% RSLogix 500 project Lab1 SLC500 3.RSS, saved by version 8.30.00.16 %
PROJECT "UNTITLED"    % processor: Bul.1763 MicroLogix 1100 Series B %

PROGRAM FILES
  LAD 2   3 rungs

DATA FILES
  O0 OUTPUT  4 elements
  I1 INPUT  6 elements
  S2 STATUS  66 elements
  B3 BINARY  1 elements
  T4 TIMER  1 elements
  C5 COUNTER  1 elements
  R6 CONTROL  1 elements
  N7 INTEGER  1 elements
  F8 FLOAT  1 elements

LADDER 2
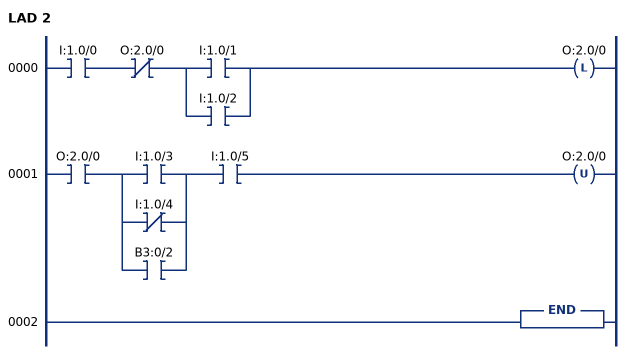
% Rung: 0 %  % edit flag set %
SOR XIC I:1.0/0 XIO O:2.0/0 BST XIC I:1.0/1 NXB XIC I:1.0/2 BND OTL O:2.0/0 EOR
% Rung: 1 %  % edit flag set %
SOR XIC O:2.0/0 BST XIC I:1.0/3 NXB XIO I:1.0/4 NXB XIC B3:0/2 BND XIC I:1.0/5 OTU O:2.0/0 EOR
% Rung: 2 %
SOR END EOR
